# EPICS substitutions: ads-ioc/valveApp/Db/valve.substitutions
global {PORT="$(PORT)"}
global {ADS_PORT="PLC_TC3"}

file "valve_vars_stream.db" {
    pattern { "P" }
        { "$(P)" }
}
